FUNCTION_BLOCK ABSTRACT OnLinkedListEventHandler EXTENDS MockEventHandler
VAR
	expectedOriginator : I_LinkedList;
END_VAR

METHOD FB_init : BOOL
VAR_INPUT
	bInitRetains : BOOL; // if TRUE, the retain variables are initialized (warm start / cold start)
	bInCopyCode : BOOL;  // if TRUE, the instance afterwards gets moved into the copy code (online change)
	ExpectedOriginator : I_LinkedList;
END_VAR
SetExpectedOriginator(ExpectedOriginator);
END_METHOD

METHOD PUBLIC SetExpectedOriginator
VAR_INPUT
	ExpectedOriginator : I_LinkedList;
END_VAR
this^.expectedOriginator := ExpectedOriginator;
END_METHOD

END_FUNCTION_BLOCK

(* stored: Version 1.1.0.1, ProductVersion 3.1.4024.12
   POU OnLinkedListEventHandler: Id {09cffca3-cc9b-4a2d-9acd-ef1bb30e4905}, SpecialFunc None
   Folder Constructor: Id {e4da78fa-81c1-4929-b0dd-c299d3677851}
   Method FB_init: Id {74de7071-4c44-4944-a2b1-4ef87701f1bf}
   Method SetExpectedOriginator: Id {200d6293-c4af-481a-9ffc-6b22f4d17f58} *)
